TYPE E_StationState :
(
	Idle := 0,
	Running := 1,
	Error := 2,
	Done := 3
) DINT;
END_TYPE

(* stored: Version 1.1.0.1, ProductVersion 3.1.4024.12
   DUT E_StationState: Id {002158df-7e10-41e2-99a1-1f8bee8e79ae} *)
